PROGRAM Main
VAR
	machine : TestMachine;
	currentState : STRING;
	start : BOOL;
	stop : BOOL;
	reset : BOOL;
	clear : BOOL;
	abort : BOOL;
END_VAR

IF start THEN
	start := FALSE;
	machine.Start();
END_IF

IF stop THEN
	stop := FALSE;
	machine.Stop();
END_IF

IF reset THEN
	reset := FALSE;
	machine.Reset();
END_IF

IF clear THEN
	clear := FALSE;
	machine.Clear();
END_IF

IF abort THEN
	abort := FALSE;
	machine.Abort();
END_IF

currentState := machine.CurrentStateName;

END_PROGRAM

(* stored: Version 1.1.0.1, ProductVersion 3.1.4024.12
   POU Main: Id {25a681c5-a485-0a21-120a-598f1114fe63}, SpecialFunc None *)
